Staubli VAL3: string.pjx

--- string.pjx ---
Parameters version=s8.13.1Cs9_BS2800 stackSize=5000 millimeterUnit=true
Program file=combineString.pgx
Program file=removeString.pgx
Program file=replacePattern.pgx
Program file=splitString.pgx
Program file=splitWord.pgx
Program file=start.pgx
Program file=stop.pgx
Program file=subString.pgx
Program file=toLowercase.pgx
Program file=toUppercase.pgx
Program file=trimString.pgx
Data file=string.dtx
Library alias=utils path=Disk://helpers/helpers.pjx
Type name=lists path=Disk://types/lists/lists.pjx

--- string.dtx ---
mdesc mNomSpeed
public lists lLists
  [0]
    string sString
string sInput[5]
lists lResult
  [0]
    string sString

--- start.pgx ---
program start()
  local num l_nElement
begin

  sInput[0] = "forward 9"
  sInput[1] = "forward 9 gtgt"
  sInput[2] = " 1878"

  call splitString(sInput, " ", lResult)

  call splitWord(sInput, lResult)

  call trimString(sInput, sResult)

  call toUppercase(sInput[1], sResult)

  call replacePattern(sInput, "r", "HGT", sResult)

  ? "## test sub: sub(sInput, 2,4,sResult)"
  call subString(sInput, 2,10,sResult)
  call utils:printStr(sResult)

   ? "## test sub: removeString(sInput, 2,3,sResult)"
  call removeString(sInput, 2,3,sResult)
  call utils:printStr(sResult)
end

--- combineString.pgx ---
public program combineString(string x_sInput)
  local num l_nElement
begin

  for l_nElement = 0 to size(x_sInput)-1
  endFor

end

--- removeString.pgx ---
public program removeString(string& x_sInput[], num x_nStart, num x_nEnd, string& x_sResult[])
  local num l_nElement
  local num l_nLength
  local string l_sLeft
  local string l_sRigt
  local string l_sRight
begin

  l_nLength = size(x_sInput)
  resize(x_sResult,1,1)
  x_sResult =""
  resize(x_sResult,1,l_nLength)

  // iterate complete input x_sInput[0] ... x_sInput[l_nLength-1]
  for l_nElement = 0 to l_nLength-1

    // ab cd efghj
    // 12 34 56789 len
    // 01 23 45678 idx
    l_sLeft = left(x_sInput[l_nElement], sel(x_nStart==0, 0, x_nStart))
    l_sRight = right(x_sInput[l_nElement], sel(len(x_sInput[l_nElement])-x_nEnd-1<0, 0, len(x_sInput[l_nElement])-x_nEnd-1))
    x_sResult[l_nElement] = l_sLeft + l_sRight

  endFor


end

--- replacePattern.pgx ---
public program replacePattern(string& x_sInput[], string x_sPattern, string x_sReplace, string& x_sResult[])
  local num l_nLength
  local num l_nElement
  local string l_sText
begin

  l_nLength = size(x_sInput)
  resize(x_sResult,1,1)
  x_sResult = ""
  resize(x_sResult,1,l_nLength)

  for l_nElement = 0 to l_nLength-1
    l_sText = x_sInput[l_nElement]
    while find(l_sText,x_sPattern)!=-1
      l_sText = replace(l_sText,x_sReplace,len(x_sPattern),find(l_sText,x_sPattern))
    endWhile
    x_sResult[l_nElement] = l_sText
  endFor

end

--- splitString.pgx ---
public program splitString(string& x_sInput[], string x_sPattern, lists& x_lResult[])
  local num l_nLength
  local num l_nElement
  local string l_sLine
  local num l_nCount
  local num l_nPos
begin

  l_nLength = size(x_sInput)
  resize(x_lResult,1,1)
  resize(x_lResult.sString,1,1)
  x_lResult.sString =""
  resize(x_lResult,1,l_nLength)

  if x_sPattern == ""
    call splitWord(x_sInput, x_lResult)
    return
  else
    // iterate complete input x_sInput[0] ... x_sInput[l_nLength-1]
    for l_nElement = 0 to l_nLength-1

      // copy element
      l_sLine = x_sInput[l_nElement]

      // search x_sPattern
      l_nCount = 0
      while len(l_sLine)!=0
        l_nPos=find(l_sLine, x_sPattern)

        if l_nPos==-1
          l_nPos=len(l_sLine)
        endIf

        if l_nCount != 0
          append(x_lResult[l_nElement].sString)
        endIf

        x_lResult[l_nElement].sString[l_nCount] = left(l_sLine,l_nPos)
        l_sLine = right(l_sLine,max(0,len(l_sLine)-l_nPos-len(x_sPattern)))
        l_nCount = l_nCount+1

      endWhile
    endFor
  endIf
end

--- splitWord.pgx ---
public program splitWord(string& x_sInput[], lists& x_lResult[])
  local num l_nLength
  local num l_nElement
  local string l_sLine
  local num l_nCount
begin

  l_nLength = size(x_sInput)
  resize(x_lResult,1,1)
  resize(x_lResult.sString,1,1)
  x_lResult.sString =""
  resize(x_lResult,1,l_nLength)

  // iterate complete input x_sInput[0] ... x_sInput[l_nLength-1]
  for l_nElement = 0 to l_nLength-1

    // copy element
    l_sLine = x_sInput[l_nElement]

    // search x_sPattern
    l_nCount = 0
    while len(l_sLine)!=0

      if l_nCount != 0
        append(x_lResult[l_nElement].sString)
      endIf

      x_lResult[l_nElement].sString[l_nCount] = left(l_sLine,1)
      l_sLine = right(l_sLine,len(l_sLine)-1)
      l_nCount = l_nCount+1

    endWhile
  endFor


end

--- subString.pgx ---
public program subString(string& x_sInput[], num x_nStart, num x_nEnd, string& x_sResult[])
  local num l_nElement
  local num l_nLength
begin

  l_nLength = size(x_sInput)
  resize(x_sResult,1,1)
  x_sResult =""
  resize(x_sResult,1,l_nLength)

  // iterate complete input x_sInput[0] ... x_sInput[l_nLength-1]
  for l_nElement = 0 to l_nLength-1

    x_sResult[l_nElement] = mid(x_sInput[l_nElement], x_nEnd-x_nStart+1,x_nStart)

  endFor

end

--- toLowercase.pgx ---
public program toLowercase(string x_sInput, string& x_sResult)
  local num l_nElement
begin
  x_sResult = ""

  for l_nElement=0 to len(x_sInput)-1
    x_sResult=x_sResult+chr(sel(asc(x_sInput,l_nElement)<65 or asc(x_sInput,l_nElement)>90,asc(x_sInput,l_nElement),asc(x_sInput,l_nElement)+32))
  endFor

end

--- toUppercase.pgx ---
public program toUppercase(string x_sInput, string& x_sResult)
  local num l_nElement
begin
  x_sResult = ""

  for l_nElement=0 to len(x_sInput)-1
    x_sResult=x_sResult+chr(sel(asc(x_sInput,l_nElement)<97 or asc(x_sInput,l_nElement)>122,asc(x_sInput,l_nElement),asc(x_sInput,l_nElement)-32))
  endFor
end

--- trimString.pgx ---
public program trimString(string& x_sInput[], string& x_sResult[])
  local num l_nLength
  local num l_nElement
  local string l_sLine
  local num l_nPos
begin

  l_nLength = size(x_sInput)
  resize(x_sResult,1,1)
  x_sResult = ""
  resize(x_sResult,1,l_nLength)

  for l_nElement = 0 to l_nLength-1

    // copy line
    l_sLine = x_sInput[l_nElement]

    while find(l_sLine," ")>=0
      l_nPos = find(l_sLine," ")
      l_sLine=delete(l_sLine,1,l_nPos)
    endWhile

    x_sResult[l_nElement] = l_sLine

  endFor

end
